INTERFACE ITF_Base

METHOD PUBLIC SetName
VAR_INPUT
	stName				: ST_BaseLabel;
END_VAR
END_METHOD

END_INTERFACE

(* stored: Version 1.1.0.1
   Itf ITF_Base: Id {303a894f-e290-0185-2c2d-0a345e19b0b8}
   Method SetName: Id {f9de5d73-0bee-0af9-32d6-cc15dbaba99a} *)
